// TIA Portal V20 export
TYPE "CS_Sides_Stations"
   STRUCT
      RL_H3_Pos : DInt;
      RR_H3_Pos : DInt;
      RL_Mid_Pos : DInt;
      RR_Mid_Pos : DInt;
      RL_H5_Pos : DInt;
      RR_H5_Pos : DInt;
      Correction : Int;
   END_STRUCT;
END_TYPE
